{attribute addProperty BoxType "IODEVICETYPE_ETHERCATPROT"}
{attribute addProperty Id "Beckhoff_EQ1xxxBeckhoff_EQ1xxx_822DEADB55469.25Beckhoff_EQ2xxxBeckhoff_EQ2xxx_ABA09D4F1871233.875Beckhoff_EQ3xxxBeckhoff_EQ3xxx_1BCF419C3460432.5SyncUnitsSyncUnits_CAB22D3B19524.375InputsInputs_C75D3FEC1280160OutputsOutputs_47D1E803848106InfoDataInfoData_E9F65A829612"}
{attribute addProperty CRC "3253249178"}
{attribute addProperty SizeInBites "8304"}
{attribute addProperty SizeInBytes "1038"}
TYPE EtherCAT_Master_EQxxxx_C1E8A49A :
STRUCT
	{attribute addProperty Name "Beckhoff_EQ1xxx"}
	Beckhoff_EQ1xxx : Beckhoff_EQ1xxx_822DEADB;
	{attribute addProperty Name "Beckhoff_EQ2xxx"}
	Beckhoff_EQ2xxx : Beckhoff_EQ2xxx_ABA09D4F;
	{attribute addProperty Name "Beckhoff_EQ3xxx"}
	Beckhoff_EQ3xxx : Beckhoff_EQ3xxx_1BCF419C;
	{attribute addProperty Name "SyncUnits"}
	SyncUnits : SyncUnits_CAB22D3B;
	{attribute addProperty Name "Inputs"}
	Inputs : Inputs_C75D3FEC;
	{attribute addProperty Name "Outputs"}
	Outputs : Outputs_47D1E803;
	{attribute addProperty Name "InfoData"}
	InfoData : InfoData_E9F65A82;
END_STRUCT
END_TYPE

(* stored: Version 1.2.0.0, ProductVersion 3.1.4024.9
   DUT EtherCAT_Master_EQxxxx_C1E8A49A: Id {a1dd021f-196b-4429-b2b3-0148eba79f65} *)
